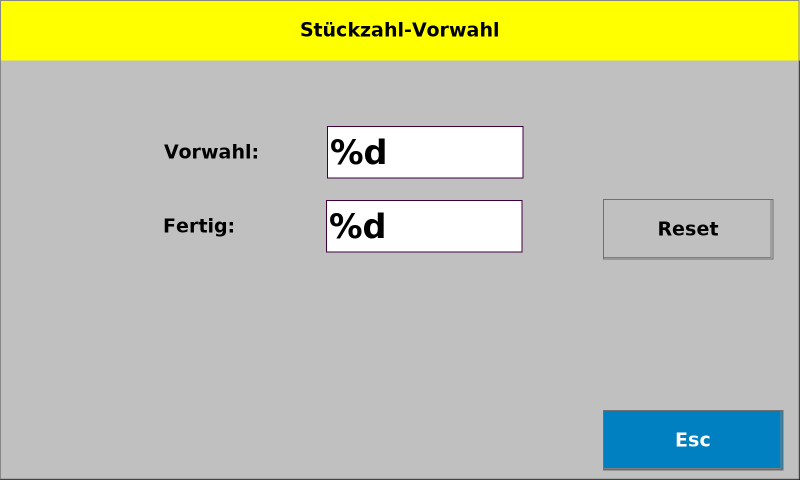
VISUALIZATION Stueckzahl  // 800x480
    Rectangle (0,0 800x480)
    Rectangle (0,0 800x60), "Stückzahl-Vorwahl"
    Button (603,410 180x60), "Esc"
        OnMouseUp: change screen: Previous 
    Rectangle (327,126 196x52), "%d", text variable: DB6.diStueck_Vorwahl
        OnMouseClick: write the text variable via VisuDialogs.Numpad, min 0, title 'Vorwahl'
    Label (161,135 159x34), "Vorwahl:"
    Rectangle (326,200 196x52), "%d", text variable: DB6.diStueck_Fertig
        OnMouseClick: write the text variable via VisuDialogs.Numpad, min 0, title 'Fertig'
    Label (160,209 159x34), "Fertig:"
    Button (603,199 170x60), "Reset"
END_VISUALIZATION

(* stored: Version 1.1.0.1, ProductVersion 3.1.4024.3
   Visu Stueckzahl: Id {cbf4d9be-7108-466d-88cb-d248112f2e32} *)
